{attribute 'GeneratedUsingTerminal: EL5001-0011-0019'}
{attribute addProperty BoxType "EL5001-0011-0019"}
{attribute addProperty Id "EtcSlaveTerminalBaseSSI_InputsAT %I*SSI_Inputs_8BC18DAC9WcStateAT %I*WcState_9091E0EB2InfoDataAT %I*InfoData_BEF6B88E18"}
{attribute addProperty CRC "4002517787"}
{attribute addProperty Size "29"}
TYPE EL5001_EE91931B EXTENDS EtcSlaveTerminalBase :
STRUCT
	{attribute addProperty Name "SSI_Inputs"}
	SSI_Inputs : SSI_Inputs_8BC18DAC;
	{attribute addProperty Name "WcState"}
	WcState : WcState_9091E0EB;
	{attribute addProperty Name "InfoData"}
	InfoData : InfoData_BEF6B88E;
END_STRUCT
END_TYPE

(* stored: Version 1.2.0.0, ProductVersion 3.1.4024.9
   DUT EL5001_EE91931B: Id {9629643e-1ced-4866-8df4-eedd83740fe4} *)
